// TIA Portal V20 export
DATA_BLOCK "InstE2MenergyMeterDriver"   // DB56
TITLE = Instanz von FB E2MenergyMeterDrv / Instance of FB E2MenergyMeterDrv
AUTHOR : SICAR
FAMILY : E2M
NAME : E2M_AIEM
VERSION : 2.0
// Energy Meter
// stored: InstanceOfName E2MenergyMeterDrv, InstanceOfType FB
"E2MenergyMeterDrv"
   // VAR_INPUT
   //    id : HW_IO := 0;
   //    firstByteData : Int := 0;
   //    connectionType : Int := 1;
   //    commResourceLimit : Int := 4;
   //    automaticUpdate : Bool := FALSE;
   //    resetMinMax : Bool := FALSE;
   //    resetEnergyCounter : Bool := FALSE;
   //    bitsConnectedHmi : Bool := FALSE;
   //    backupCycleEnCount : Time := T#5S;
   // END_VAR
   // VAR_OUTPUT
   //    timeBetweenUpdate : Time := T#0MS;
   //    timeBetweenUpdateMax : Time := T#0MS;
   //    timeStampMeasValues : DTL := DTL#1970-01-01-00:00:00;
   //    driverData { ExternalAccessible := 'False'; ExternalVisible := 'False'; ExternalWritable := 'False'} : "LSicar_typeEnMeterVisuStruct";
   //    energyCounter { ExternalAccessible := 'False'; ExternalVisible := 'False'; ExternalWritable := 'False'} : "typeEnCounter";
   //    errorCode : DWord := 16#0000_0000;
   //    errorLocation : Word := 16#0000;
   //    timeStampEnCount : DTL := DTL#1970-01-01-00:00:00;
   // END_VAR
   // VAR_IN_OUT
   //    bitsHmi : "typeEnMeterBits";
   //    commResourceCounter : Int := 0;
   // END_VAR
   // VAR
   //    instReadDataRecord { S7_SetPoint := 'True'} : RDREC;
   //    instWriteDataRecord { S7_SetPoint := 'True'} : WRREC;
   //    instEnCountUpdateTimer { S7_SetPoint := 'True'} : TON_TIME;
   //    instTimeMeasurement { S7_SetPoint := 'True'} : TON_TIME;
   //    instWatchdog { S7_SetPoint := 'True'} : TON_TIME;
   //    statInputVariablesOk : Bool := FALSE;
   //    statResetEnCountRequest : Bool := FALSE;
   //    statReadDataRecRequest : Bool := FALSE;
   //    statWriteDataRecRequest : Bool := FALSE;
   //    statRestoreEnergy : Bool := FALSE;
   //    statStartAcyclicHmiOld : Bool := FALSE;
   //    statResetEnergyHmiOld : Bool := FALSE;
   //    statResetEnergyOld : Bool := FALSE;
   //    statResetMinMaxHmiOld : Bool := FALSE;
   //    statResetMinMaxOld : Bool := FALSE;
   //    statRunUpdateTimer : Bool := FALSE;
   //    statWatchdogRun : Bool := FALSE;
   //    statUserDataVariant : Byte := 16#00;
   //    statSmState : Int := 0;
   //    statSmStateNext : Int := 0;
   //    statReadRecIndex : Int := 0;
   //    statReadRecMaxLength : UInt := 0;
   //    statTimetoUpdate : Time := T#0MS;
   //    statVmeasurementValues : "typeEnMeterValues";
   //    statVenergyCounter : "typeEnMeterCounter";
   //    statBitsInternalHmi : "typeEnMeterBits";
   // END_VAR
   // VAR RETAIN
   //    statRestoreEnCountValues : "typeEnMeterRestore";
   // END_VAR
   // VAR
   //    statAuxTimeBetweenUpdateMax { S7_SetPoint := 'True'} : Time := T#0MS;
   //    statErrorCode { ExternalVisible := 'False'} : DWord := 16#0000_0000;
   // END_VAR
BEGIN
   driverData.uL1L2 := 480.6464;
   driverData.uL2L3 := 479.3329;
   driverData.uL3L1 := 482.4024;
   driverData.uL1 := 277.0244;
   driverData.uL2 := 283.0648;
   driverData.uL3 := 272.9026;
   driverData.uL1L2Min := 470.1363;
   driverData.uL2L3Min := 469.0945;
   driverData.uL3L1Min := 472.4617;
   driverData.uL1Min := 271.5103;
   driverData.uL2Min := 277.1332;
   driverData.uL3Min := 267.6445;
   driverData.uL1L2Max := 486.0269;
   driverData.uL2L3Max := 484.8441;
   driverData.uL3L1Max := 487.8807;
   driverData.uL1Max := 280.1993;
   driverData.uL2Max := 286.2231;
   driverData.uL3Max := 276.0547;
   driverData.uPhPhAverage := 480.7939;
   driverData.uPhNaverage := 277.6639;
   driverData.uPhPhAverageMin := 470.5642;
   driverData.uPhNaverageMin := 272.105;
   driverData.uPhPhAverageMax := 486.2456;
   driverData.uPhNaverageMax := 280.8176;
   driverData.iL1 := 0.6297245;
   driverData.iL2 := 0.4116209;
   driverData.iL3 := 0.4021624;
   driverData.iL1Min := 0.5503862;
   driverData.iL2Min := 0.3512777;
   driverData.iL3Min := 0.3410119;
   driverData.iL1Max := 2.701323;
   driverData.iL2Max := 2.376321;
   driverData.iL3Max := 1.768756;
   driverData.iAverage := 0.4811693;
   driverData.iAverageMin := 0.4219982;
   driverData.iAverageMax := 2.194234;
   driverData.f := 59.99327;
   driverData.fMin := 59.9567;
   driverData.fMax := 60.07609;
   driverData.sTotal := 400.7156;
   driverData.sTotalMin := 349.7767;
   driverData.sTotalMax := 1823.43;
   driverData.pTotal := 277.3849;
   driverData.pTotalMin := 220.7085;
   driverData.pTotalMax := 670.0833;
   driverData.qTotal := -19.24654;
   driverData.qTotalMin := -422.0206;
   driverData.qTotalMax := -5.418034;
   driverData.cosL1 := 0.8610036;
   driverData.cosL1Min := 0.3576268;
   driverData.cosL1Max := 0.9157406;
   driverData.cosL2 := 0.5061908;
   driverData.cosL2Min := 0.05827232;
   driverData.cosL2Max := 0.7094496;
   driverData.cosL3 := 0.6214478;
   driverData.cosL3Min := 0.1665398;
   driverData.cosL3Max := 0.7301649;
   driverData.cosAverage := 0.6922238;
   driverData.cosAverageMin := 0.2474333;
   driverData.cosAverageMax := 0.7716895;
   driverData.sL1 := 174.449;
   driverData.sL2 := 116.5154;
   driverData.sL3 := 109.7511;
   driverData.sL1Min := 151.7066;
   driverData.sL2Min := 99.03358;
   driverData.sL3Min := 92.7289;
   driverData.sL1Max := 744.3881;
   driverData.sL2Max := 669.9091;
   driverData.sL3Max := 480.3434;
   driverData.pL1 := 150.2012;
   driverData.pL2 := 58.97903;
   driverData.pL3 := 68.20461;
   driverData.pL1Min := 127.6866;
   driverData.pL2Min := 20.87;
   driverData.pL3Min := 52.5906;
   driverData.pL1Max := 281.8818;
   driverData.pL2Max := 194.1828;
   driverData.pL3Max := 220.8245;
   driverData.qL1 := -4.041785;
   driverData.qL2 := 41.25737;
   driverData.qL3 := -56.46213;
   driverData.qL1Min := -144.4171;
   driverData.qL2Min := -98.00859;
   driverData.qL3Min := -198.8008;
   driverData.qL1Max := 28.71266;
   driverData.qL2Max := 50.3845;
   driverData.qL3Max := -53.43742;
   driverData.eActiveRate1Import := 736796.1;
   driverData.eActiveRate2Import := 0.0;
   driverData.eActiveRate1Export := 0.0002530577;
   driverData.eActiveRate2Export := 0.0;
   driverData.eReactiveRate1Import := 5676.457;
   driverData.eReactiveRate2Import := 0.0;
   driverData.eReactiveRate1Export := 293593.3;
   driverData.eReactiveRate2Export := 0.0;
   driverData.eApparentRate1Import := 1470773.0;
   driverData.eApparentRate2Import := 0.0;
   driverData.rTimeDataEnergy := DTL#1970-01-01-00:00:00;
   driverData.rTimeDataValue := DTL#1970-01-01-00:00:00;
   driverData.uPhPhMod := 16#0000;
   driverData.uPhNmod := 16#0000;
   driverData.iMod := 16#0000;
   driverData.sMod := 16#0000;
   driverData.pMod := 16#0000;
   driverData.qMod := 16#0000;
   driverData.eMod := 16#0000;
   driverData.fMod := 16#0000;
   driverData.cosMod := 16#0000;
   driverData.calculateValue1 := 16#0000;
   driverData.calculateValue2 := 16#0000;
   driverData.calculateValue3 := 16#0000;
   driverData.calculateValue4 := 16#0000;
   driverData.calculateValue5 := 16#0000;
   driverData.calculateValue6 := 16#0000;
   driverData.energyMeterUnit := 16#0000;
   driverData.restStartAuto := FALSE;
   driverData.readValue := FALSE;
   driverData.connectionType := 0;
   driverData.driverError := 0;
   energyCounter.activeRate1Imp := 0.0;
   energyCounter.activeRate1Exp := 0.0;
   energyCounter.activeRate2Imp := 0.0;
   energyCounter.activeRate2Exp := 0.0;
   energyCounter.reactiveRate1Imp := 0.0;
   energyCounter.reactiveRate1Exp := 0.0;
   energyCounter.reactiveRate2Imp := 0.0;
   energyCounter.reactiveRate2Exp := 0.0;
   energyCounter.apparentRate1Imp := 0.0;
   energyCounter.apparentRate2Imp := 0.0;
   instReadDataRecord.REQ := FALSE;
   instReadDataRecord.ID := 0;
   instReadDataRecord.INDEX := 0;
   instReadDataRecord.MLEN := 0;
   instReadDataRecord.VALID := FALSE;
   instReadDataRecord.BUSY := FALSE;
   instReadDataRecord.ERROR := FALSE;
   instReadDataRecord.STATUS := 16#0000_0000;
   instReadDataRecord.LEN := 0;
   instWriteDataRecord.REQ := FALSE;
   instWriteDataRecord.ID := 0;
   instWriteDataRecord.INDEX := 0;
   instWriteDataRecord.LEN := 0;
   instWriteDataRecord.DONE := FALSE;
   instWriteDataRecord.BUSY := FALSE;
   instWriteDataRecord.ERROR := FALSE;
   instWriteDataRecord.STATUS := 16#0000_0000;
   instEnCountUpdateTimer.PT := T#0MS;
   instEnCountUpdateTimer.IN := FALSE;
   instTimeMeasurement.PT := T#0MS;
   instTimeMeasurement.IN := FALSE;
   instWatchdog.PT := T#0MS;
   instWatchdog.IN := FALSE;
   statVmeasurementValues.dataRecordVersion := 16#00;
   statVmeasurementValues.reserved := 16#00;
   statVmeasurementValues.voltageL1N := 0.0;
   statVmeasurementValues.voltageL2N := 0.0;
   statVmeasurementValues.voltageL3N := 0.0;
   statVmeasurementValues.voltageL1L2 := 0.0;
   statVmeasurementValues.voltageL2L3 := 0.0;
   statVmeasurementValues.voltageL3L1 := 0.0;
   statVmeasurementValues.currentL1 := 0.0;
   statVmeasurementValues.currentL2 := 0.0;
   statVmeasurementValues.currentL3 := 0.0;
   statVmeasurementValues.powerFactorL1 := 0.0;
   statVmeasurementValues.powerFactorL2 := 0.0;
   statVmeasurementValues.powerFactorL3 := 0.0;
   statVmeasurementValues.powerFactorOverall := 0.0;
   statVmeasurementValues.frequency := 0.0;
   statVmeasurementValues.voltageSymmetry := 0.0;
   statVmeasurementValues.currentSymmetry := 0.0;
   statVmeasurementValues.apparentPowerL1 := 0.0;
   statVmeasurementValues.apparentPowerL2 := 0.0;
   statVmeasurementValues.apparentPowerL3 := 0.0;
   statVmeasurementValues.apparentPowerOverall := 0.0;
   statVmeasurementValues.reactivePowerL1 := 0.0;
   statVmeasurementValues.reactivePowerL2 := 0.0;
   statVmeasurementValues.reactivePowerL3 := 0.0;
   statVmeasurementValues.reactivePowerOverall := 0.0;
   statVmeasurementValues.effectivePowerL1 := 0.0;
   statVmeasurementValues.effectivePowerL2 := 0.0;
   statVmeasurementValues.effectivePowerL3 := 0.0;
   statVmeasurementValues.effectivePowerOverall := 0.0;
   statVmeasurementValues.phaseAngleL1 := 0.0;
   statVmeasurementValues.phaseAngleL2 := 0.0;
   statVmeasurementValues.phaseAngleL3 := 0.0;
   statVmeasurementValues.appEnOverall32bit := 0.0;
   statVmeasurementValues.reaEnOverall32bit := 0.0;
   statVmeasurementValues.effEnOverall32bit := 0.0;
   statVmeasurementValues.reaEnImport32bit := 0.0;
   statVmeasurementValues.reaEnExport32bit := 0.0;
   statVmeasurementValues.effEnImport32bit := 0.0;
   statVmeasurementValues.effEnExport32bit := 0.0;
   statVmeasurementValues.appEnOverall64bit := 0.0;
   statVmeasurementValues.reaEnOverall64bit := 0.0;
   statVmeasurementValues.effEnOverall64bit := 0.0;
   statVmeasurementValues.reaEnImport64bit := 0.0;
   statVmeasurementValues.reaEnExport64bit := 0.0;
   statVmeasurementValues.effEnImport64bit := 0.0;
   statVmeasurementValues.effEnExport64bit := 0.0;
   statVenergyCounter.dataRecordVersion := 16#00;
   statVenergyCounter.reserved := 16#00;
   statVenergyCounter.controlByte1L1 := 16#00;
   statVenergyCounter.controlByte2L1 := 16#00;
   statVenergyCounter.controlByte1L2 := 16#00;
   statVenergyCounter.controlByte2L2 := 16#00;
   statVenergyCounter.controlByte1L3 := 16#00;
   statVenergyCounter.controlByte2L3 := 16#00;
   statVenergyCounter.effEnImportL1 := 0.0;
   statVenergyCounter.effEnExportL1 := 0.0;
   statVenergyCounter.reaEnImportL1 := 0.0;
   statVenergyCounter.reaEnExportL1 := 0.0;
   statVenergyCounter.appEnL1 := 0.0;
   statVenergyCounter.effEnImportL2 := 0.0;
   statVenergyCounter.effEnExportL2 := 0.0;
   statVenergyCounter.reaEnImportL2 := 0.0;
   statVenergyCounter.reaEnExportL2 := 0.0;
   statVenergyCounter.appEnL2 := 0.0;
   statVenergyCounter.effEnImportL3 := 0.0;
   statVenergyCounter.effEnExportL3 := 0.0;
   statVenergyCounter.reaEnImportL3 := 0.0;
   statVenergyCounter.reaEnExportL3 := 0.0;
   statVenergyCounter.appEnL3 := 0.0;
   statBitsInternalHmi.startAcyclic := FALSE;
   statBitsInternalHmi.startAuto := FALSE;
   statBitsInternalHmi.resetMinMaxData := FALSE;
   statBitsInternalHmi.resetEnergyMeter := FALSE;
   statRestoreEnCountValues.dataRecordVersion := 16#00;
   statRestoreEnCountValues.reserved := 16#00;
   statRestoreEnCountValues.controlByte1L1 := 16#00;
   statRestoreEnCountValues.controlByte2L1 := 16#00;
   statRestoreEnCountValues.controlByte1L2 := 16#00;
   statRestoreEnCountValues.controlByte2L2 := 16#00;
   statRestoreEnCountValues.controlByte1L3 := 16#00;
   statRestoreEnCountValues.controlByte2L3 := 16#00;
   statRestoreEnCountValues.effEnImportL1 := 0.0;
   statRestoreEnCountValues.effEnExportL1 := 0.0;
   statRestoreEnCountValues.reaEnImportL1 := 0.0;
   statRestoreEnCountValues.reaEnExportL1 := 0.0;
   statRestoreEnCountValues.appEnL1 := 0.0;
   statRestoreEnCountValues.effEnImportL2 := 0.0;
   statRestoreEnCountValues.effEnExportL2 := 0.0;
   statRestoreEnCountValues.reaEnImportL2 := 0.0;
   statRestoreEnCountValues.reaEnExportL2 := 0.0;
   statRestoreEnCountValues.appEnL2 := 0.0;
   statRestoreEnCountValues.effEnImportL3 := 0.0;
   statRestoreEnCountValues.effEnExportL3 := 0.0;
   statRestoreEnCountValues.reaEnImportL3 := 0.0;
   statRestoreEnCountValues.reaEnExportL3 := 0.0;
   statRestoreEnCountValues.appEnL3 := 0.0;
END_DATA_BLOCK
